// TIA Portal V19 export
FUNCTION_BLOCK "Block_3"   // FB2, LAD
{ S7_Optimized_Access := 'TRUE' }
// stored: MemoryReserve 100, SetENOAutomatically false
BEGIN
END_FUNCTION_BLOCK
